
// ===== library: MasterCopy "Copy of Program blocks in gw_material_parameters" =====

// folder: gw_material_parameters

DATA_BLOCK "db_gw_material_parameters"   // DB950
{ S7_Optimized_Access := 'TRUE' }
VERSION : 0.1
   VAR RETAIN
      subsystem_1 : "udt_gw_subsystem_1";
      subsystem_2 : "udt_gw_subsystem_2";
   END_VAR
   VAR
      valid_overall : Bool;   // Gesamt gültig / overall valid
      difference_overall : Bool;   // Gesamt differenz / overall difference
      accept_overall : Bool;   // Gesamt übernehmen / Accept overall
      reject_overall : Bool;   // Gesamt verwerfen / Reject overall
      save_overall : Bool;   // Gesamt in Datenbank speichern / Save overall to Getzner database
      save_overall_ok : Bool;   // Rueckmeldung von Getzner speichern erfolgreich / Getzner save successfull
   END_VAR
BEGIN
END_DATA_BLOCK

FUNCTION "fc_gw_material_parameters" : Void   // FC950, FBD
{ S7_Optimized_Access := 'TRUE' }
VERSION : 0.1
   VAR_IN_OUT
      subsystem_1 : "udt_gw_subsystem_1";
      subsystem_2 : "udt_gw_subsystem_2";
   END_VAR
   VAR_TEMP
      fault_unable_to_save : Bool;
   END_VAR
BEGIN

REGION Network 1: Sollwerte Grenzen prüfen / Check setpoint limits
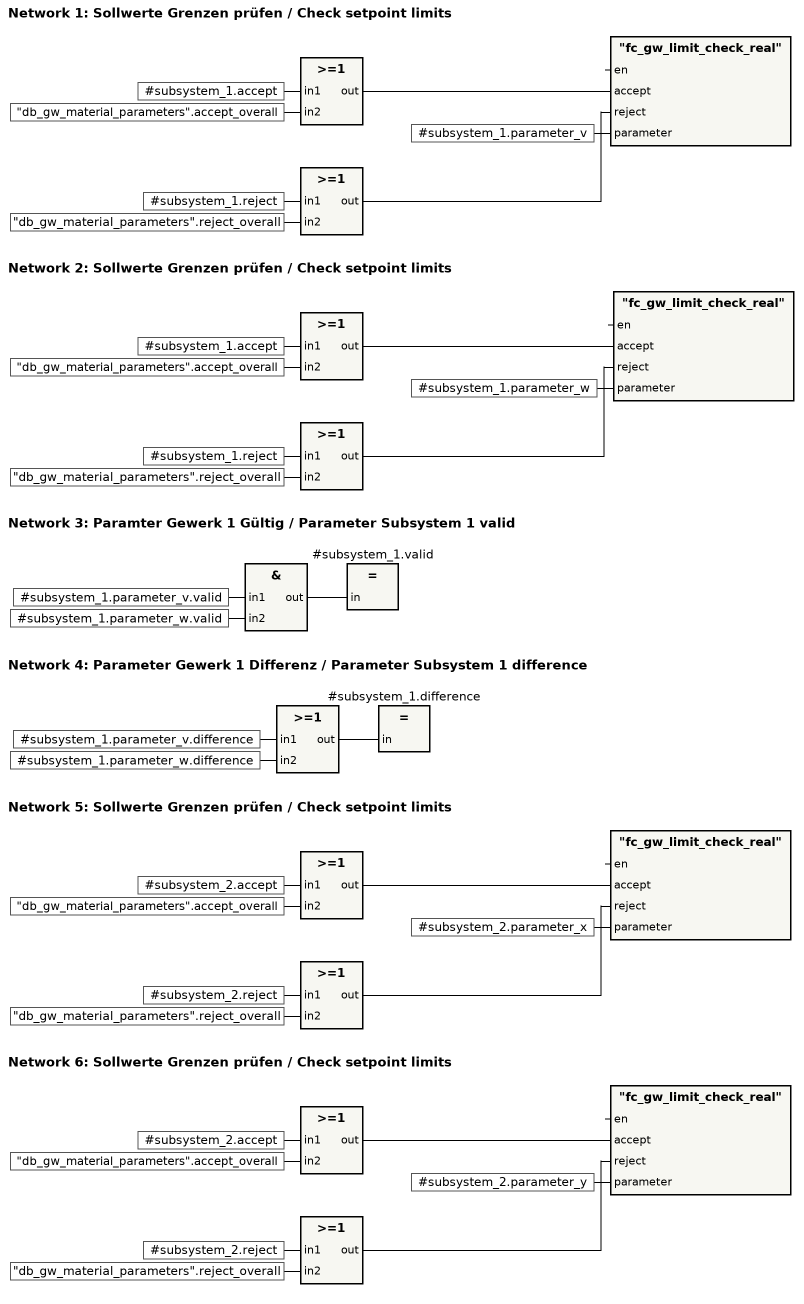
   "fc_gw_limit_check_real"(accept := #subsystem_1.accept OR "db_gw_material_parameters".accept_overall,
                           reject := #subsystem_1.reject OR "db_gw_material_parameters".reject_overall,
                           parameter := #subsystem_1.parameter_v);
END_REGION

REGION Network 2: Sollwerte Grenzen prüfen / Check setpoint limits
   "fc_gw_limit_check_real"(accept := #subsystem_1.accept OR "db_gw_material_parameters".accept_overall,
                           reject := #subsystem_1.reject OR "db_gw_material_parameters".reject_overall,
                           parameter := #subsystem_1.parameter_w);
END_REGION

REGION Network 3: Paramter Gewerk 1 Gültig / Parameter Subsystem 1 valid
   #subsystem_1.valid := #subsystem_1.parameter_v.valid AND #subsystem_1.parameter_w.valid;
END_REGION

REGION Network 4: Parameter Gewerk 1 Differenz / Parameter Subsystem 1 difference
   #subsystem_1.difference := #subsystem_1.parameter_v.difference OR #subsystem_1.parameter_w.difference;
END_REGION

REGION Network 5: Sollwerte Grenzen prüfen / Check setpoint limits
   "fc_gw_limit_check_real"(accept := #subsystem_2.accept OR "db_gw_material_parameters".accept_overall,
                           reject := #subsystem_2.reject OR "db_gw_material_parameters".reject_overall,
                           parameter := #subsystem_2.parameter_x);
END_REGION

REGION Network 6: Sollwerte Grenzen prüfen / Check setpoint limits
   "fc_gw_limit_check_real"(accept := #subsystem_2.accept OR "db_gw_material_parameters".accept_overall,
                           reject := #subsystem_2.reject OR "db_gw_material_parameters".reject_overall,
                           parameter := #subsystem_2.parameter_y);
END_REGION

REGION Network 7: Sollwerte Grenzen prüfen / Check setpoint limits
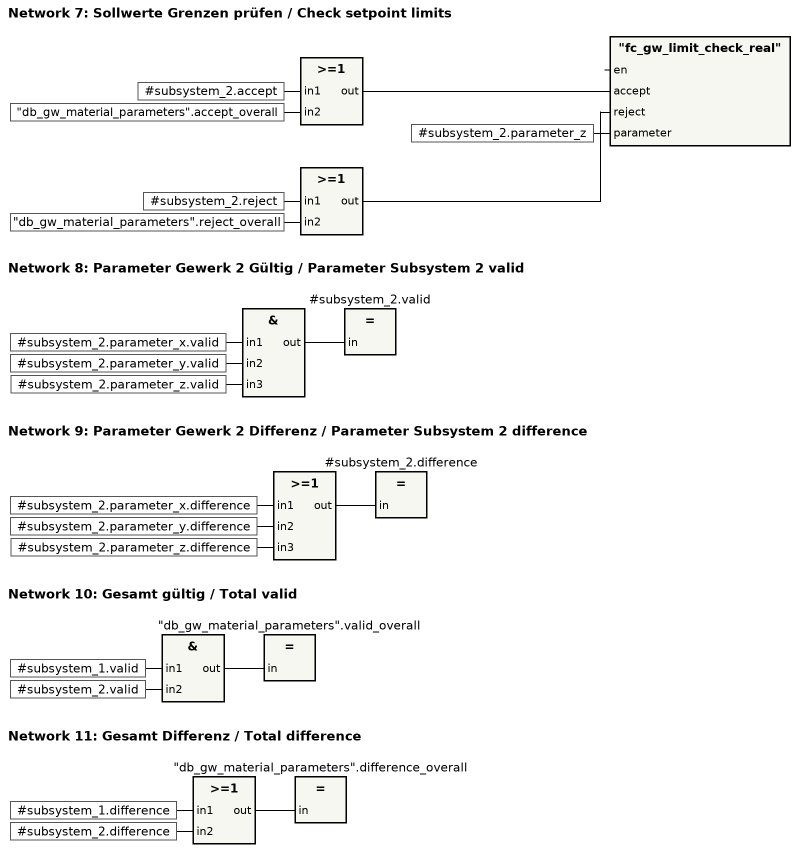
   "fc_gw_limit_check_real"(accept := #subsystem_2.accept OR "db_gw_material_parameters".accept_overall,
                           reject := #subsystem_2.reject OR "db_gw_material_parameters".reject_overall,
                           parameter := #subsystem_2.parameter_z);
END_REGION

REGION Network 8: Parameter Gewerk 2 Gültig / Parameter Subsystem 2 valid
   #subsystem_2.valid := #subsystem_2.parameter_x.valid AND #subsystem_2.parameter_y.valid AND #subsystem_2.parameter_z.valid;
END_REGION

REGION Network 9: Parameter Gewerk 2 Differenz / Parameter Subsystem 2 difference
   #subsystem_2.difference := #subsystem_2.parameter_x.difference OR #subsystem_2.parameter_y.difference OR #subsystem_2.parameter_z.difference;
END_REGION

REGION Network 10: Gesamt gültig / Total valid
   "db_gw_material_parameters".valid_overall := #subsystem_1.valid AND #subsystem_2.valid;
END_REGION

REGION Network 11: Gesamt Differenz / Total difference
   "db_gw_material_parameters".difference_overall := #subsystem_1.difference OR #subsystem_2.difference;
END_REGION

REGION Network 12 (SCL): Übernehmen und Verwerfen rücksetzen / Reset accept and reject
   #subsystem_1.accept:= FALSE;
   #subsystem_1.reject:= FALSE;
   #subsystem_2.accept:= FALSE;
   #subsystem_2.reject:= FALSE;
   "db_gw_material_parameters".accept_overall:= FALSE;
   "db_gw_material_parameters".reject_overall:= FALSE;
END_REGION

REGION Network 13 (SCL): Gesamt in Getzner Datenbank abspeichern / Save total to Getzner database
   "ton_fault_save_system".TON(IN:="db_gw_material_parameters".save_overall,
                                     PT:=t#5s);

   IF ("db_gw_material_parameters".save_overall AND
       (NOT "db_gw_material_parameters".valid_overall OR
       "db_gw_material_parameters".difference_overall)) OR
       "ton_fault_save_system".Q THEN
       #fault_unable_to_save := TRUE;  //---------- create HMI Message ---------
       "db_gw_material_parameters".save_overall := FALSE;
   END_IF;

   IF "db_gw_material_parameters".save_overall_ok THEN
       "db_gw_material_parameters".save_overall := FALSE;
       "db_gw_material_parameters".save_overall_ok := FALSE;
   END_IF;
END_REGION
END_FUNCTION

FUNCTION "fc_gw_limit_check_real" : Void   // FC951, FBD
{ S7_Optimized_Access := 'TRUE' }
VERSION : 0.1
   VAR_INPUT
      accept : Bool;
      reject : Bool;
   END_VAR
   VAR_IN_OUT
      parameter : "udt_gw_parameters";
   END_VAR
BEGIN

REGION Network 1 (SCL): Gueltig / Valid
   IF #parameter.value > #parameter.max OR
       #parameter.value < #parameter.min THEN
       #parameter.valid:= FALSE;
   ELSE
       #parameter.valid:= TRUE;
   END_IF;
END_REGION

REGION Network 2 (SCL): Differenz zwischen Aktiv / Difference to active value
   IF #parameter.value <> #parameter.active_value THEN
       #parameter.difference:= TRUE;
   ELSE
       #parameter.difference:= FALSE;
   END_IF;
END_REGION

REGION Network 3 (SCL): Uebernehmen Verwerfen / Accept / reject
   IF #parameter.valid AND #accept THEN
       #parameter.active_value:= #parameter.value;
   END_IF;

   IF #reject THEN
       #parameter.value:= #parameter.active_value;
   END_IF;
END_REGION
END_FUNCTION

// ===== library: MasterCopy "udt_gw_parameters" =====

TYPE "udt_gw_parameters"
   STRUCT
      value : Real;   // Parameterwert der auf der Visu eingegeben wird / Parameter value entered via HMI
      active_value : Real;   // Parameterwert mit dem die Anlage arbeitet / Parameter value used by the system
      min : Real;   // Min Begrenzung / Minimum limit
      max : Real;   // Max Begrenzung / Maximum limit
      valid : Bool;   // Eingabewert Befindet sich innerhalb der Grenzwerte Min Max / Input value is within min/max limits
      difference : Bool;   // Differenz zu aktiv / Difference to active value
   END_STRUCT;
END_TYPE

// ===== library: MasterCopy "udt_gw_subsystem_1" =====

TYPE "udt_gw_subsystem_1"
   STRUCT
      parameter_v : "udt_gw_parameters";
      parameter_w : "udt_gw_parameters";
      valid : Bool;   // Gewerk gültig / Subsystem valid
      difference : Bool;   // Gewerk differenz zu Aktiv / Subsystem difference to active value
      accept : Bool;   // Gewerk übernehmen / Accept Subsystem
      reject : Bool;   // Gewerk verwerfen / Reject Subsystem
   END_STRUCT;
END_TYPE

// ===== library: MasterCopy "udt_gw_subsystem_2" =====

TYPE "udt_gw_subsystem_2"
   STRUCT
      parameter_x : "udt_gw_parameters";
      parameter_y : "udt_gw_parameters";
      parameter_z : "udt_gw_parameters";
      valid : Bool;   // Gewerk gültig / Subsystem valid
      difference : Bool;   // Gewerk differenz zu Aktiv / Subsystem difference to active value
      accept : Bool;   // Gewerk übernehmen / Accept Subsystem
      reject : Bool;   // Gewerk verwerfen / Reject Subsystem
   END_STRUCT;
END_TYPE